// TIA Portal V20 export
TYPE "typeIdentRfHmi"
// stored: Access Published
   STRUCT
      selectedUnit : USInt;
      selectedEM : USInt;
      rfReaderId : USInt;   // RF Reader ID
      numberOfRf : USInt;   // Number of used RFIDs
      rfReader : Array[0.."NO_OF_RF_IDENT_DEVICES"] of "LSicar_typeIdentInterfaceHmi";   // RF Reader
   END_STRUCT;
END_TYPE
